(* PLC project Trafic_Light, Unknown Unnamed 1 *)
(* stored: creationDateTime 2020-10-12T21:33:17, modificationDateTime 2024-02-07T14:34:37 *)

PROGRAM Trafic_light
  VAR
    TOF0 : TOF;
    TOF1 : TOF;
    TOF2 : TOF;
  END_VAR
  VAR
    O_LEDRed AT %QX0.0 : BOOL;  (* red LED on pin 14 *)
    O_LEDOrange AT %QX0.1 : BOOL;  (* orange LED on pin 15 *)
    O_LEDGreen AT %QX0.2 : BOOL;  (* Green LED on pin 16 *)
    First_cycle AT %QX0.3 : BOOL := TRUE;  (* Is true only during the first scan cycle *)
  END_VAR
  VAR
    F_TRIG0 : F_TRIG;
    F_TRIG1 : F_TRIG;
    F_TRIG2 : F_TRIG;
  END_VAR

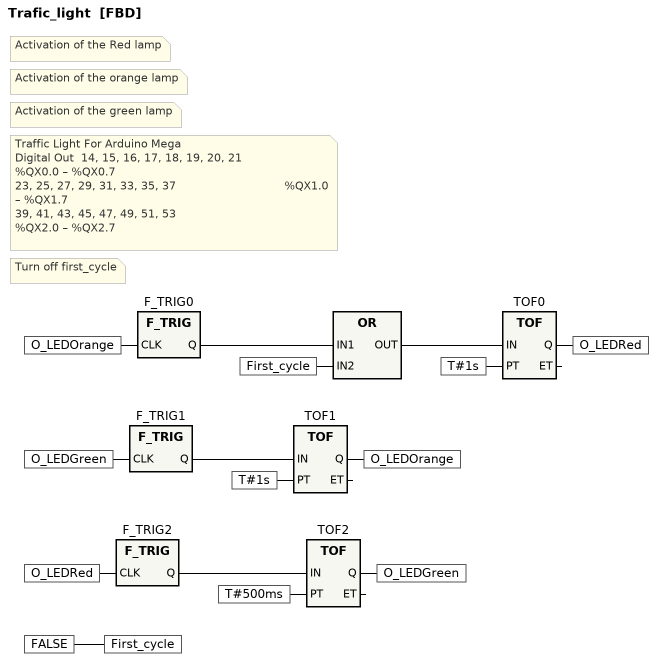
(* FBD diagram, written out as Structured Text *)
(* Traffic Light For Arduino Mega


Digital Out	14, 15, 16, 17, 18, 19, 20, 21                    %QX0.0 – %QX0.7
23, 25, 27, 29, 31, 33, 35, 37                               %QX1.0 – %QX1.7
39, 41, 43, 45, 47, 49, 51, 53	                               %QX2.0 – %QX2.7 *)
(* Activation of the Red lamp *)
F_TRIG0(CLK := O_LEDOrange);
TOF0(IN := F_TRIG0.Q OR First_cycle, PT := T#1s);
O_LEDRed := TOF0.Q;
(* Activation of the orange lamp *)
F_TRIG1(CLK := O_LEDGreen);
TOF1(IN := F_TRIG1.Q, PT := T#1s);
O_LEDOrange := TOF1.Q;
(* Activation of the green lamp *)
F_TRIG2(CLK := O_LEDRed);
TOF2(IN := F_TRIG2.Q, PT := T#500ms);
O_LEDGreen := TOF2.Q;
(* Turn off first_cycle *)
First_cycle := FALSE;
END_PROGRAM

CONFIGURATION Config0
  RESOURCE Res0 ON PLC
    TASK task0(INTERVAL := T#20ms, PRIORITY := 0);
    PROGRAM instance0 WITH task0 : Trafic_light;
  END_RESOURCE
END_CONFIGURATION
